PROGRAM PRG_BreakfastTask
VAR
	Ready : BOOL;
END_VAR

CASE GVL_MorningRoutine.State_Breakfast OF

    0: // Idle
        IF GVL_MorningRoutine.StartBreakfast THEN
            GVL_MorningRoutine.State_Breakfast := 10;
        END_IF

    10: // Wait for Task 1 to finish
        Ready := IsReady(GVL_MorningRoutine.ReadyForBreakfast);
        IF Ready THEN
            GVL_MorningRoutine.State_Breakfast := 20;
        END_IF

    20: // Make breakfast
        GVL_MorningRoutine.MakingBreakfast := TRUE;
        GVL_MorningRoutine.State_Breakfast := 30;

    30: // Eat breakfast
        GVL_MorningRoutine.EatingBreakfast := TRUE;
        GVL_MorningRoutine.ReadyToLeave := TRUE;
        GVL_MorningRoutine.State_Breakfast := 40;

    40: // Done
        // Task completed

END_CASE

END_PROGRAM

(* stored: Version 1.1.0.1, ProductVersion 3.1.4024.15
   POU PRG_BreakfastTask: Id {e5b94054-dba6-4d30-8fd2-4e1bd4eee6f0}, SpecialFunc None *)
